  [4496] = {x=916.926, y=-64.508, z=44, rx=-180, rz=142.794, shoulder=lefty, elbow=epositive, wrist=wpositive, fatherId=fReference[0]}
  [4497] = {x=918.172, y=-63.562, z=44, rx=180, rz=142.766, shoulder=lefty, elbow=epositive, wrist=wpositive, fatherId=fReference[0]}
  [4498] = {x=919.418, y=-62.615, z=44, rx=-180, rz=142.738, shoulder=lefty, elbow=epositive, wrist=wpositive, fatherId=fReference[0]}
  [4499] = {x=920.664, y=-61.667, z=44, rx=-180, rz=142.71, shoulder=lefty, elbow=epositive, wrist=wpositive, fatherId=fReference[0]}
  [4500] = {x=921.91, y=-60.719, z=44, rx=-180, rz=142.683, shoulder=lefty, elbow=epositive, wrist=wpositive, fatherId=fReference[0]}
  [4501] = {x=923.155, y=-59.769, z=44, rx=-180, rz=142.657, shoulder=lefty, elbow=epositive, wrist=wpositive, fatherId=fReference[0]}
  [4502] = {x=924.4, y=-58.82, z=44, rx=180, rz=142.631, shoulder=lefty, elbow=epositive, wrist=wpositive, fatherId=fReference[0]}
  [4503] = {x=925.644, y=-57.869, z=44, rx=-180, rz=142.605, shoulder=lefty, elbow=epositive, wrist=wpositive, fatherId=fReference[0]}
  [4504] = {x=926.889, y=-56.918, z=44, rx=180, rz=142.58, shoulder=lefty, elbow=epositive, wrist=wpositive, fatherId=fReference[0]}
  [4505] = {x=928.133, y=-55.966, z=44, rx=-180, rz=142.555, shoulder=lefty, elbow=epositive, wrist=wpositive, fatherId=fReference[0]}
  [4506] = {x=929.377, y=-55.013, z=44, rx=180, rz=142.53, shoulder=lefty, elbow=epositive, wrist=wpositive, fatherId=fReference[0]}
  [4507] = {x=930.621, y=-54.06, z=44, rx=-180, rz=142.507, shoulder=lefty, elbow=epositive, wrist=wpositive, fatherId=fReference[0]}
  [4508] = {x=931.864, y=-53.106, z=44, rx=-180, rz=142.483, shoulder=lefty, elbow=epositive, wrist=wpositive, fatherId=fReference[0]}
  [4509] = {x=933.107, y=-52.152, z=44, rx=-180, rz=142.46, shoulder=lefty, elbow=epositive, wrist=wpositive, fatherId=fReference[0]}
  [4510] = {x=934.35, y=-51.197, z=44, rx=-180, rz=142.437, shoulder=lefty, elbow=epositive, wrist=wpositive, fatherId=fReference[0]}
  [4511] = {x=935.593, y=-50.241, z=44, rx=180, rz=142.415, shoulder=lefty, elbow=epositive, wrist=wpositive, fatherId=fReference[0]}
  [4512] = {x=936.835, y=-49.284, z=44, rx=180, rz=142.393, shoulder=lefty, elbow=epositive, wrist=wpositive, fatherId=fReference[0]}
  [4513] = {x=938.078, y=-48.328, z=44, rx=180, rz=142.372, shoulder=lefty, elbow=epositive, wrist=wpositive, fatherId=fReference[0]}
  [4514] = {x=939.32, y=-47.37, z=44, rx=180, rz=142.351, shoulder=lefty, elbow=epositive, wrist=wpositive, fatherId=fReference[0]}
  [4515] = {x=940.561, y=-46.412, z=44, rx=180, rz=142.331, shoulder=lefty, elbow=epositive, wrist=wpositive, fatherId=fReference[0]}
  [4516] = {x=941.803, y=-45.454, z=44, rx=-180, rz=142.311, shoulder=lefty, elbow=epositive, wrist=wpositive, fatherId=fReference[0]}
  [4517] = {x=943.044, y=-44.494, z=44, rx=180, rz=142.291, shoulder=lefty, elbow=epositive, wrist=wpositive, fatherId=fReference[0]}
  [4518] = {x=944.286, y=-43.535, z=44, rx=-180, rz=142.272, shoulder=lefty, elbow=epositive, wrist=wpositive, fatherId=fReference[0]}
  [4519] = {x=945.527, y=-42.575, z=44, rx=180, rz=142.254, shoulder=lefty, elbow=epositive, wrist=wpositive, fatherId=fReference[0]}
  [4520] = {x=946.768, y=-41.614, z=44, rx=-180, rz=142.235, shoulder=lefty, elbow=epositive, wrist=wpositive, fatherId=fReference[0]}
  [4521] = {x=948.008, y=-40.653, z=44, rx=180, rz=142.217, shoulder=lefty, elbow=epositive, wrist=wpositive, fatherId=fReference[0]}
  [4522] = {x=949.249, y=-39.691, z=44, rx=180, rz=142.2, shoulder=lefty, elbow=epositive, wrist=wpositive, fatherId=fReference[0]}
  [4523] = {x=950.489, y=-38.729, z=44, rx=-180, rz=142.183, shoulder=lefty, elbow=epositive, wrist=wpositive, fatherId=fReference[0]}
  [4524] = {x=951.729, y=-37.767, z=44, rx=180, rz=142.167, shoulder=lefty, elbow=epositive, wrist=wpositive, fatherId=fReference[0]}
  [4525] = {x=952.969, y=-36.804, z=44, rx=180, rz=142.151, shoulder=lefty, elbow=epositive, wrist=wpositive, fatherId=fReference[0]}
  [4526] = {x=954.209, y=-35.841, z=44, rx=180, rz=142.135, shoulder=lefty, elbow=epositive, wrist=wpositive, fatherId=fReference[0]}
  [4527] = {x=955.448, y=-34.877, z=44, rx=180, rz=142.12, shoulder=lefty, elbow=epositive, wrist=wpositive, fatherId=fReference[0]}
  [4528] = {x=956.688, y=-33.913, z=44, rx=-180, rz=142.105, shoulder=lefty, elbow=epositive, wrist=wpositive, fatherId=fReference[0]}
  [4529] = {x=957.927, y=-32.948, z=44, rx=180, rz=142.09, shoulder=lefty, elbow=epositive, wrist=wpositive, fatherId=fReference[0]}
  [4530] = {x=959.166, y=-31.983, z=44, rx=180, rz=142.076, shoulder=lefty, elbow=epositive, wrist=wpositive, fatherId=fReference[0]}
  [4531] = {x=960.405, y=-31.018, z=44, rx=-180, rz=142.063, shoulder=lefty, elbow=epositive, wrist=wpositive, fatherId=fReference[0]}
  [4532] = {x=961.644, y=-30.052, z=44, rx=180, rz=142.05, shoulder=lefty, elbow=epositive, wrist=wpositive, fatherId=fReference[0]}
  [4533] = {x=962.882, y=-29.086, z=44, rx=180, rz=142.037, shoulder=lefty, elbow=epositive, wrist=wpositive, fatherId=fReference[0]}
  [4534] = {x=964.121, y=-28.12, z=44, rx=180, rz=142.025, shoulder=lefty, elbow=epositive, wrist=wpositive, fatherId=fReference[0]}
  [4535] = {x=965.359, y=-27.153, z=44, rx=180, rz=142.013, shoulder=lefty, elbow=epositive, wrist=wpositive, fatherId=fReference[0]}
  [4536] = {x=966.598, y=-26.186, z=44, rx=180, rz=142.002, shoulder=lefty, elbow=epositive, wrist=wpositive, fatherId=fReference[0]}
  [4537] = {x=967.836, y=-25.219, z=44, rx=180, rz=141.991, shoulder=lefty, elbow=epositive, wrist=wpositive, fatherId=fReference[0]}
  [4538] = {x=969.074, y=-24.251, z=44, rx=180, rz=141.98, shoulder=lefty, elbow=epositive, wrist=wpositive, fatherId=fReference[0]}
  [4539] = {x=970.312, y=-23.283, z=44, rx=180, rz=141.97, shoulder=lefty, elbow=epositive, wrist=wpositive, fatherId=fReference[0]}
  [4540] = {x=971.55, y=-22.315, z=44, rx=180, rz=141.96, shoulder=lefty, elbow=epositive, wrist=wpositive, fatherId=fReference[0]}
  [4541] = {x=972.787, y=-21.347, z=44, rx=-180, rz=141.951, shoulder=lefty, elbow=epositive, wrist=wpositive, fatherId=fReference[0]}
  [4542] = {x=974.025, y=-20.378, z=44, rx=180, rz=141.942, shoulder=lefty, elbow=epositive, wrist=wpositive, fatherId=fReference[0]}
  [4543] = {x=975.263, y=-19.409, z=44, rx=180, rz=141.934, shoulder=lefty, elbow=epositive, wrist=wpositive, fatherId=fReference[0]}
  [4544] = {x=976.5, y=-18.44, z=44, rx=-180, rz=141.926, shoulder=lefty, elbow=epositive, wrist=wpositive, fatherId=fReference[0]}
  [4545] = {x=977.737, y=-17.471, z=44, rx=-180, rz=141.918, shoulder=lefty, elbow=epositive, wrist=wpositive, fatherId=fReference[0]}
  [4546] = {x=978.975, y=-16.501, z=44, rx=-180, rz=141.911, shoulder=lefty, elbow=epositive, wrist=wpositive, fatherId=fReference[0]}
  [4547] = {x=980.212, y=-15.532, z=44, rx=180, rz=141.904, shoulder=lefty, elbow=epositive, wrist=wpositive, fatherId=fReference[0]}
  [4548] = {x=981.449, y=-14.562, z=44, rx=-180, rz=141.898, shoulder=lefty, elbow=epositive, wrist=wpositive, fatherId=fReference[0]}
  [4549] = {x=982.686, y=-13.592, z=44, rx=-180, rz=141.892, shoulder=lefty, elbow=epositive, wrist=wpositive, fatherId=fReference[0]}
  [4550] = {x=983.923, y=-12.621, z=44, rx=180, rz=141.887, shoulder=lefty, elbow=epositive, wrist=wpositive, fatherId=fReference[0]}
  [4551] = {x=985.16, y=-11.651, z=44, rx=180, rz=141.882, shoulder=lefty, elbow=epositive, wrist=wpositive, fatherId=fReference[0]}
  [4552] = {x=986.397, y=-10.681, z=44, rx=-180, rz=141.877, shoulder=lefty, elbow=epositive, wrist=wpositive, fatherId=fReference[0]}
  [4553] = {x=987.634, y=-9.71, z=44, rx=180, rz=141.873, shoulder=lefty, elbow=epositive, wrist=wpositive, fatherId=fReference[0]}
  [4554] = {x=988.87, y=-8.739, z=44, rx=180, rz=141.869, shoulder=lefty, elbow=epositive, wrist=wpositive, fatherId=fReference[0]}
  [4555] = {x=990.107, y=-7.769, z=44, rx=-180, rz=141.866, shoulder=lefty, elbow=epositive, wrist=wpositive, fatherId=fReference[0]}
  [4556] = {x=991.344, y=-6.798, z=44, rx=180, rz=141.863, shoulder=lefty, elbow=epositive, wrist=wpositive, fatherId=fReference[0]}
  [4557] = {x=992.58, y=-5.827, z=44, rx=180, rz=141.86, shoulder=lefty, elbow=epositive, wrist=wpositive, fatherId=fReference[0]}
  [4558] = {x=993.817, y=-4.856, z=44, rx=180, rz=141.858, shoulder=lefty, elbow=epositive, wrist=wpositive, fatherId=fReference[0]}
  [4559] = {x=995.054, y=-3.885, z=44, rx=180, rz=141.857, shoulder=lefty, elbow=epositive, wrist=wpositive, fatherId=fReference[0]}
  [4560] = {x=996.29, y=-2.914, z=44, rx=-180, rz=141.855, shoulder=lefty, elbow=epositive, wrist=wpositive, fatherId=fReference[0]}
  [4561] = {x=997.527, y=-1.942, z=44, rx=180, rz=141.854, shoulder=lefty, elbow=epositive, wrist=wpositive, fatherId=fReference[0]}
  [4562] = {x=998.763, y=-0.971, z=44, rx=180, rz=141.854, shoulder=lefty, elbow=epositive, wrist=wpositive, fatherId=fReference[0]}
  [4563] = {x=1000, z=44, rx=-180, rz=141.854, shoulder=lefty, elbow=epositive, wrist=wpositive, fatherId=fReference[0]}
public tool tTool = {z=600, rz=-125, fatherId=flange[0], ioLink=valve1}
public num kk
public bool spd_cntl
public mdesc cnst_vel = {tmax=100, rmax=100, leave=0.1, reach=0.1, blend=cartesian}
public jointRx Jnt_cnfg = {j3=90, j5=90, j6=90}
public num Ref_Vel
sio sioASCII = {link=Socket\trsf_sv}
public bool check_status
aio Tpompe = {link=CanIO\RemIO\remio0_QW}
dio doValve1 = {link=valve1}
dio doValve2 = {link=valve2}
dio doPompe = {link=CanIO\RemIO\remio0_Q}

--- start.pgx ---
public program start()
  local num ID_val
begin
   disablePower()
  cls()
  userPage()
  title(" Concrete 3D Printer-Linear Path ")
  putln("Written by Erfan.")
  setProfile("Manual","123")
  if getProfile() == "Manual"
    putln("Profile is set to Remote Control.")
  endIf
  delay(3)
  enablePower()
  if(watch(isPowered(),3) == false)
    putln("Arm power supply cannot be swithced on.")
  endIf
  putln("Arm power is now switched on.")
  delay(3)
  taskCreate "Initialization",1,init_prgm()
  putln("Pump has been launched.")
  putln("Nozzle is closed.")
  delay(2)
  ID_val = 0.75
  //taskCreate "SocketOpening",10,open_socket()
  //taskCreate "CheckComnunic",20,check_cmt()
  //wait(check_status == true)
  //delay(2)
  //taskCreate "DataReading",40,read_data()
  //taskCreate "MotionControl",40,motion_cntl()
  //taskCreate "DataDisplay",40,show_data()
  //taskCreate "DataSending",50,send_data()


  /////////////////////////////////////
  // Stop Printing
  call stop_print()

  //***************************************

  // Go to configuration
  spd_cntl = false
  resetMotion()
  setMonitorSpeed(10)
  movej(Jnt_cnfg[0],tTool[0],cnst_vel[0])
  waitEndMove()

  //**************************************************

  // Go to Start point - 1st Layer
  spd_cntl = false
  setMonitorSpeed(10)
  movej(jJoint[0],tTool[0],cnst_vel[0])
  movel(pPoint[0],tTool[0],cnst_vel[0])
  movel(pPoint[1],tTool[0],cnst_vel[0])
  waitEndMove()


  // Printing - 1st Layer
  setProfile("Automatic","123")
  spd_cntl = true
  resetMotion()

   // Starting printing
  call launch_print()

  for kk = 3 to 1519 step 1
    setMoveId(0)
    movel(pPoint[kk],tTool[0],mNomSpeed[0])
    wait(getMoveId() >= ID_val)
  endFor

  // Stop Printing
  call stop_print()

  //**************************************************

  // Go to Start point - 2nd Layer
  resetMotion()
  setProfile("Manual","123")
  spd_cntl = false
  resetMotion()
  setMonitorSpeed(100)
  movel(pPoint[1520],tTool[0],cnst_vel[0])
  movel(pPoint[1521],tTool[0],cnst_vel[0])
  movel(pPoint[1522],tTool[0],cnst_vel[0])
  movel(pPoint[1523],tTool[0],cnst_vel[0])
  waitEndMove()

  // Printing - 2nd Layer
  setProfile("Automatic","123")
  spd_cntl = true
  resetMotion()

   // Starting printing
  call launch_print()

  for kk = 1525 to 3041 step 1
    setMoveId(0)
    movel(pPoint[kk],tTool[0],mNomSpeed[0])
    wait(getMoveId() >= ID_val)
  endFor

  // Stop Printing
  call stop_print()

  //******************************************

  // Go to Start point - 3rd Layer

  resetMotion()
  setProfile("Manual","123")
  spd_cntl = false
  resetMotion()
  setMonitorSpeed(100)
  movel(pPoint[3042],tTool[0],cnst_vel[0])
  movel(pPoint[3042],tTool[0],cnst_vel[0])
  movel(pPoint[3043],tTool[0],cnst_vel[0])
  movel(pPoint[3044],tTool[0],cnst_vel[0])
  movel(pPoint[3045],tTool[0],cnst_vel[0])
  waitEndMove()


  // Printing - 3rd Layer
  setProfile("Automatic","123")
  spd_cntl = true
  resetMotion()

  // Starting printing
  call launch_print()

  for kk = 3047 to 4563 step 1
    setMoveId(0)
    movel(pPoint[kk],tTool[0],mNomSpeed[0])
    wait(getMoveId() >= ID_val)
  endFor

 // Stop Printing
  call stop_print()

  //**************************************************


  ///////////////////////////
  cls()
  userPage()
  title(" Concrete 3D Printer-Linear Path ")
  putln("printing procedure has been finished.")

  // Go to configuration
  setProfile("Manual","123")
  spd_cntl = false
  resetMotion()
  setMonitorSpeed(100)
  movej(Jnt_cnfg[0],tTool[0],cnst_vel[0])
  waitEndMove()


  /////////////////////

  stopMove()
  disablePower()


  ///////////////////////////////////////////




end

--- open_socket.pgx ---
public program open_socket()
begin

  sioCtrl(sioASCII,"port",11002)
  //sioCtrl(sioASCII,"port",1002)
  //sioCtrl(sioASCII,"target","10.3.1.185")
  //sioCtrl(sioASCII,"target","10.10.5.1")
  sioCtrl(sioASCII,"target","169.254.209.1")
  sioCtrl(sioASCII,"timeout",10)
  sioCtrl(sioASCII,"endOfString",13)
  sioCtrl(sioASCII,"nangle",true)

  putln(" ")
  putln("The communication socket is open.")

  check_status = false

end

--- read_ID.pgx ---
program read_ID()
begin
  do

    putln(getMoveId())
    ID_val = getMoveId()

  until check_ID != true
end
